Universal Robots PolyScope program: test straight weld.urp

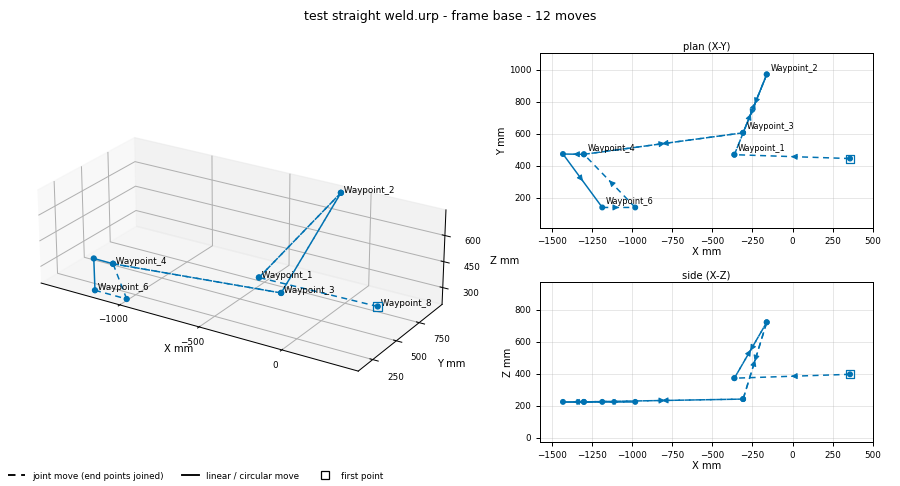
[picture p0: tool path of test straight weld.urp in frame base, 12 of 12 moves have a stored position in this frame; points joined in program order, loops and branches not executed]
Program test straight weld (installation=default directory=/programs createdIn=5.14.5 lastSavedIn=5.14.5 robotSerialNumber=20236801216)
Calibrated DH parameters: a=[-0.000021, -0.748897, -0.28186, -0.00004, -0.000055, 0]; d=[0.236225, -424.082933, -1564.66872, 1988.95162, 0.159094, 0.153873]; alpha=[1.570844, 0.001002, 0.000337, 1.571488, -1.569996, 0]; deltaTheta=[0, -0.516316, 5.626292, 1.173211, 0.000001, 0]
InitVariablesNode
Robot Program (runOnlyOnce=true)
  SafeHome (positionOptionType=SPEED_AND_ACCELERATION speed=1.047198 acceleration=1.396263 nextMotionTime=2)
  MoveJ speed 60 deg/s, acceleration 80 deg/s^2 (useActiveTCP=true) feature=Base
    Waypoint Waypoint_8: TCP in base x=359.082 y=445.186 z=397.106 mm, rx=1.9529 ry=2.2906 rz=0.1872 rad; joints [-182.315, -117.852, 126.735, -13.011, -11.421, -6.036] deg; TCP offset x=-5.053 y=-331.71 z=103.574 mm, rx=1.2092 ry=-1.2092 rz=1.2092 rad
  'extrude out a foot'
  URCap WireTank Serial (WireTank Serial, WireTank, LLC) dataModel(byte_array=true, NODE_TITLE=Serial Bridge uR1, Command=[252,82,49], QUERY=false, OUTPUT_ENTRY=Static, Variable(key=OUTPUT_VARIABLE, variable(name=HwResp)))
  Wait Sleep waitTime=48
  URCap WireTank Serial (WireTank Serial, WireTank, LLC) dataModel(QUERY=false, NODE_TITLE=Serial Bridge uR0, Command=[252,82,48], byte_array=true, OUTPUT_ENTRY=Static, Variable(key=OUTPUT_VARIABLE, variable=HwResp))
  Popup Message (haltProgram=false message=grab extrusion then press ok inputType=Text)
  'approach'
  MoveJ speed 60 deg/s, acceleration 80 deg/s^2 (useActiveTCP=true) feature=Base
    Waypoint Waypoint_1: TCP in base x=-363.139 y=469.335 z=372.923 mm, rx=0.3211 ry=3.1107 rz=0.1051 rad; joints [-102.381, -94.177, 139.921, 99.856, 0.714, -149.503] deg
    Waypoint Waypoint_2: TCP in base x=-161.023 y=970.525 z=722.063 mm, rx=-0.5549 ry=0.1065 rz=0.3286 rad; joints [-74.514, -75.395, 129.709, 210.687, -169.172, 54.348] deg
    Waypoint Waypoint_3: TCP in base x=-308.534 y=606.018 z=242.406 mm, rx=1.3698 ry=1.0668 rz=-1.2572 rad; joints [-84.909, -52.754, 88.074, 55.223, 94.97, 14.302] deg
    Waypoint Waypoint_4: TCP in base x=-1302.622 y=471.672 z=225 mm, rx=1.8756 ry=0.6001 rz=-1.8483 rad; joints [-42.019, -35.832, 56.335, 69.976, 90.58, 102.09] deg; TCP offset x=-5.053 y=-331.71 z=103.574 mm, rx=1.2092 ry=-1.2092 rz=1.2092 rad
  'get into position'
  MoveL speed 20 mm/s, acceleration 100 mm/s^2 (useActiveTCP=true) feature=Base
    Waypoint Waypoint_5: TCP in base x=-1433.412 y=473.471 z=225 mm, rx=1.8753 ry=0.6037 rz=-1.8523 rad; joints [-38.295, -25.763, 35.633, 80.393, 90.555, 105.858] deg; TCP offset x=-5.053 y=-331.71 z=103.574 mm, rx=1.2092 ry=-1.2092 rz=1.2092 rad
  'preheat'
  Wait Sleep waitTime=8
  'extrude'
  URCap WireTank Serial (WireTank Serial, WireTank, LLC) dataModel(byte_array=true, NODE_TITLE=Serial Bridge uR1, Command=[252,82,49], QUERY=false, OUTPUT_ENTRY=Static, Variable(key=OUTPUT_VARIABLE, variable=HwResp))
  Wait Sleep waitTime=0.1
  MoveL speed 10 mm/s, acceleration 50 mm/s^2 (useActiveTCP=true) feature=Base
    Waypoint Waypoint_6: TCP in base x=-1188.017 y=139.835 z=225 mm, rx=1.8748 ry=0.6043 rz=-1.8518 rad; joints [-31.683, -51.736, 87.639, 54.429, 90.534, 112.423] deg; TCP offset x=-5.053 y=-331.71 z=103.574 mm, rx=1.2092 ry=-1.2092 rz=1.2092 rad
  URCap WireTank Serial (WireTank Serial, WireTank, LLC) dataModel(QUERY=false, NODE_TITLE=Serial Bridge uR0, Command=[252,82,48], byte_array=true, OUTPUT_ENTRY=Static, Variable(key=OUTPUT_VARIABLE, variable=HwResp))
  MoveJ speed 60 deg/s, acceleration 80 deg/s^2 (useActiveTCP=true) feature=Base
    Waypoint Waypoint_7: TCP in base x=-982.135 y=139.822 z=225 mm, rx=1.8748 ry=0.6043 rz=-1.8518 rad; joints [-39.635, -61.764, 106.155, 45.862, 90.59, 104.473] deg; TCP offset x=-5.053 y=-331.71 z=103.574 mm, rx=1.2092 ry=-1.2092 rz=1.2092 rad
  'go back'
  MoveJ speed 60 deg/s, acceleration 80 deg/s^2 (useActiveTCP=true) feature=Base
    Waypoint Waypoint_4: TCP in base x=-1302.622 y=471.672 z=225 mm, rx=1.8756 ry=0.6001 rz=-1.8483 rad; joints [-42.019, -35.832, 56.335, 69.976, 90.58, 102.09] deg; TCP offset x=-5.053 y=-331.71 z=103.574 mm, rx=1.2092 ry=-1.2092 rz=1.2092 rad
    Waypoint Waypoint_3: TCP in base x=-308.534 y=606.018 z=242.406 mm, rx=1.3698 ry=1.0668 rz=-1.2572 rad; joints [-84.909, -52.754, 88.074, 55.223, 94.97, 14.302] deg; TCP offset x=-5.053 y=-331.71 z=103.574 mm, rx=1.2092 ry=-1.2092 rz=1.2092 rad
    Waypoint Waypoint_2: TCP in base x=-161.023 y=970.525 z=722.063 mm, rx=-0.5549 ry=0.1065 rz=0.3286 rad; joints [-74.514, -75.395, 129.709, 210.687, -169.172, 54.348] deg
    Waypoint Waypoint_1: TCP in base x=-363.139 y=469.335 z=372.923 mm, rx=0.3211 ry=3.1107 rz=0.1051 rad; joints [-102.381, -94.177, 139.921, 99.856, 0.714, -149.503] deg
  SafeHome (positionOptionType=SPEED_AND_ACCELERATION speed=1.047198 acceleration=1.396263 nextMotionTime=2)
